Fanuc KAREL source: kb00195.KL

-- PROVISIONAL review KL for V770-1; original PC SHA256 23b37c38f9bfe8c5f94b2ff2471500cac0505e4a8044d4c3c8f77d68b3ed73e8
-- Incomplete behavior may be omitted. Consult companion uncertainty JSON. Do not deploy.
PROGRAM KB00195
%NOLOCKGROUP
BEGIN
  -- UNRESOLVED_PC offsets 5-14; opcodes 3F,75
  -- UNRESOLVED_PC offsets 19-28; opcodes 3F,75
  -- UNRESOLVED_PC offsets 33-40; opcodes 9D,23
  -- UNRESOLVED_PC offsets 45-52; opcodes 9D,23
  -- UNRESOLVED_PC offsets 57-64; opcodes 9D,23
  -- UNRESOLVED_PC offsets 69-76; opcodes 9D,23
  -- UNRESOLVED_PC offsets 81-88; opcodes 9D,23
  -- UNRESOLVED_PC offsets 93-149; opcodes 27,22,2A,22,2A,22,22,22,22,22,22,31
  -- UNRESOLVED_PC offsets 154-158; opcodes 7F
END KB00195
